FUNCTION_BLOCK F_LREAL_TO_BYTE (* convert LREAL to BYTE *)
  (* Standard: 61131-3; Classification: type conversion function *)
  (* Version 0.0, 2013-08-29, 4DIAC-IDE, 4DIAC-Consortium *)
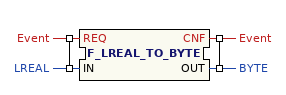
  EVENT_INPUT
    REQ WITH IN; (* Service Request *)
  END_EVENT
  EVENT_OUTPUT
    CNF WITH OUT; (* Confirmation of Requested Service *)
  END_EVENT
  VAR_INPUT
    IN : LREAL; (* input value *)
  END_VAR
  VAR_OUTPUT
    OUT : BYTE; (* output value *)
  END_VAR
  (* Service APPLICATION/RESOURCE: convert LREAL to BYTE *)
END_FUNCTION_BLOCK
